PROGRAM MAIN
VAR
	//stTestInstance : ST_Event;
	bBoolean : BOOL := FALSE;
	
	eEventType1 : E_EventType := E_EventType.Alarm;
	eEventSeverity1 : TcEventSeverity := TcEventSeverity.Critical;
	nEventIdentity1 : UDINT := 42;
	sEventText1: STRING(255) := 'spooky event';
	
	EventLogger : EventLogger;
END_VAR

(*IF NOT bBoolean THEN
	UpdateEventTimeStampWithSystemTime(stEvent := stTestInstance);
	bBoolean := TRUE;
END_IF *)

IF bBoolean THEN
	EventLogger.AddEvent(eEventType1, eEventSeverity1, nEventIdentity1, sEventText1);
	bBoolean := FALSE;
END_IF

END_PROGRAM

(* stored: Version 1.1.0.1, ProductVersion 3.1.4024.5
   POU MAIN: Id {7229c79b-ffb5-4a7c-9e41-6545460c70da}, SpecialFunc None *)
